FUNCTION_BLOCK PnPVacuum (* Basic Function Block Type *)
  (* Standard: 61499-2 *)
  (* Version 0.0, 2/7/2012, XPMUser, nxtControl GmbH, Template *)
  PACKAGE Main;
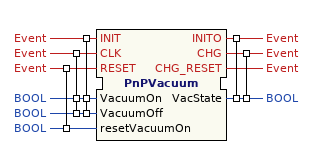
  EVENT_INPUT
    INIT WITH VacuumOn, VacuumOff; (* Initialization Request *)
    CLK WITH VacuumOn, VacuumOff; (* Clock signal *)
    RESET WITH resetVacuumOn;
  END_EVENT
  EVENT_OUTPUT
    INITO WITH VacState; (* Initialization Confirm *)
    CHG WITH VacState; (* Execution Confirmation *)
    CHG_RESET;
  END_EVENT
  VAR_INPUT
    VacuumOn : BOOL; (* Input event qualifier *)
    VacuumOff : BOOL;
    resetVacuumOn : BOOL;
  END_VAR
  VAR_OUTPUT
    VacState : BOOL; (* State of vacuum *)
  END_VAR
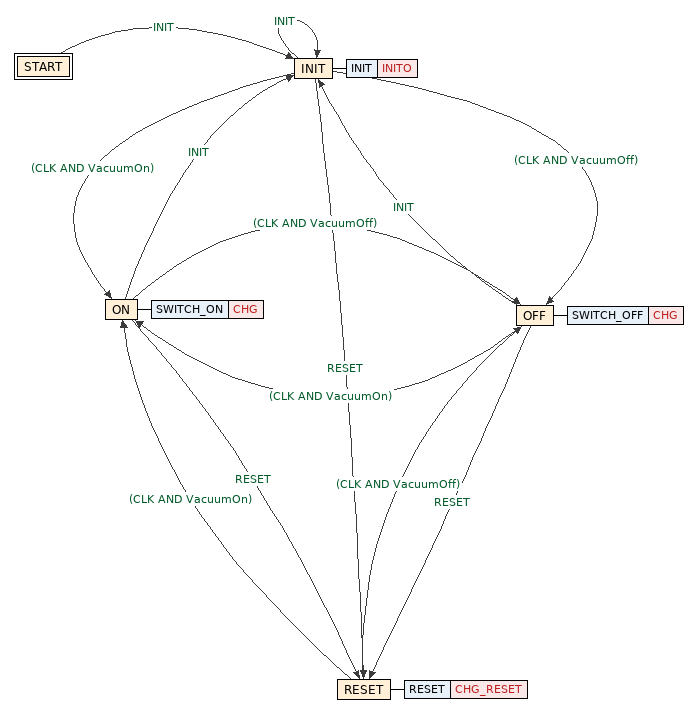
  EC_STATES
    START; (* Initial State *)
    INIT : INIT -> INITO; (* Initialization *)
    ON : SWITCH_ON -> CHG; (* Normal execution *)
    OFF : SWITCH_OFF -> CHG;
    RESET : RESET -> CHG_RESET;
  END_STATES
  EC_TRANSITIONS
    START TO INIT := INIT;
    INIT TO OFF := (CLK AND VacuumOff);
    OFF TO ON := (CLK AND VacuumOn);
    ON TO OFF := (CLK AND VacuumOff);
    INIT TO ON := (CLK AND VacuumOn);
    ON TO INIT := INIT;
    OFF TO INIT := INIT;
    INIT TO INIT := INIT;
    OFF TO RESET := RESET;
    ON TO RESET := RESET;
    INIT TO RESET := RESET;
    RESET TO OFF := (CLK AND VacuumOff);
    RESET TO ON := (CLK AND VacuumOn);
  END_TRANSITIONS
  ALGORITHM INIT IN ST: (* Initialization algorithm *)
INIT:=FALSE;
IF VacuumOn = TRUE THEN
  VacState := TRUE;
ELSIF VacuumOff = TRUE THEN
  VacState := FALSE;
END_IF;
  END_ALGORITHM
  ALGORITHM SWITCH_ON IN ST:
VacState := TRUE;
  END_ALGORITHM
  ALGORITHM SWITCH_OFF IN ST:
VacState := FALSE;
  END_ALGORITHM
  ALGORITHM RESET IN ST:
VacState:=resetVacuumOn;
  END_ALGORITHM
END_FUNCTION_BLOCK
